{attribute 'linkalways'} 
{attribute 'no_explicit_call' := 'This FB is a CLASS and must be accessed using methods or properties'}
{attribute 'enable_dynamic_creation'}
FUNCTION_BLOCK Node_F_VN_FillContainer_TcVnVector3_SINT EXTENDS VisionNode
VAR
    ipContainer : _ITcVnContainer;
    aValue : _TcVnVector3_SINT;
    hrPrev : _HRESULT(S_OK);
    hresult : _HRESULT(S_OK);
END_VAR

METHOD PUBLIC  Clone : I_Node
VAR
    pNode : POINTER TO Node_F_VN_FillContainer_TcVnVector3_SINT;
END_VAR
pNode := __NEW(Node_F_VN_FillContainer_TcVnVector3_SINT);
Clone := pNode^;
END_METHOD

METHOD FB_init : BOOL
VAR_INPUT
    bInitRetains : BOOL; // if TRUE, the retain variables are initialized (warm start / cold start)
    bInCopyCode : BOOL;  // if TRUE, the instance afterwards gets moved into the copy code (online change)
END_VAR
AddInput('ipContainer', ipContainer);
AddInput('aValue', aValue);
AddInput('hrPrev', hrPrev);
AddOutput('ipContainer', ipContainer);
AddOutput('hresult',hresult);
END_METHOD

METHOD PROTECTED OnExecute
hresult.Value := F_VN_FillContainer_TcVnVector3_SINT(
    ipContainer := ipContainer.Value,
    aValue := aValue.Value,
    hrPrev:= hrPrev.Value);
END_METHOD

METHOD PUBLIC PreExecutionCheck
VAR_INPUT
    Check : I_PreExecutionChecks;
END_VAR
Check.IsTrue(ipContainer.IsValid, 'ipContainer must be a valid container');
Check.IsTrue(ipContainer.IsType(TC_GLOBAL_CONST_LIST.ContainerType_Vector_TcVnVector3_SINT), 'ipContainer contains incorrect type');
END_METHOD

END_FUNCTION_BLOCK

(* stored: Version 1.1.0.1, ProductVersion 3.1.4026.13
   POU Node_F_VN_FillContainer_TcVnVector3_SINT: Id {6cae267d-5c29-4fca-a8ec-2f0a14e1d38c}, SpecialFunc None
   Folder Constructor: Id {91221916-3144-49e1-afeb-9c1e2f6e3ae5}
   Method Clone: Id {20ff1215-67ec-4d7a-a1e6-13db0724bd96}
   Method FB_init: Id {6db19bec-ace2-4928-a0e5-1933f7247393}
   Method OnExecute: Id {c066047f-a50a-415c-860b-02aeb0c54818}
   Method PreExecutionCheck: Id {3eead35e-1037-46c0-bac7-80737598d984} *)
